{attribute 'linkalways'} 
{attribute 'no_explicit_call' := 'This FB is a CLASS and must be accessed using methods or properties'}
{attribute 'enable_dynamic_creation'}
FUNCTION_BLOCK Node_F_VN_MedianElementElementwise_SINT EXTENDS VisionNode
VAR
    ipContainer : _ITcVnContainer;
    nMedian : _SINT(0);
    hrPrev : _HRESULT(S_OK);
    hresult : _HRESULT(S_OK);
END_VAR

METHOD PUBLIC  Clone : I_Node
VAR
	pNode : POINTER TO Node_F_VN_MedianElementElementwise_SINT;
END_VAR
pNode := __NEW(Node_F_VN_MedianElementElementwise_SINT);
Clone := pNode^;
END_METHOD

METHOD FB_init : BOOL
VAR_INPUT
	bInitRetains : BOOL; // if TRUE, the retain variables are initialized (warm start / cold start)
	bInCopyCode : BOOL;  // if TRUE, the instance afterwards gets moved into the copy code (online change)
END_VAR
AddInput('ipContainer', ipContainer);
AddInput('nMedian', nMedian);
AddInput('hrPrev', hrPrev);
AddOutput('ipContainer', ipContainer);
AddOutput('hresult',hresult);
END_METHOD

METHOD PROTECTED OnExecute : HRESULT
hresult.Value := F_VN_MedianElementElementwise_SINT(
    ipContainer := ipContainer.Value,
    nMedian := nMedian.Value,
    hrPrev:= hrPrev.Value);
END_METHOD

METHOD PUBLIC PreExecutionCheck
VAR_INPUT
	Check : I_PreExecutionChecks;
END_VAR
Check.IsTrue(ipContainer.IsValid, 'ipContainer must be a valid container');
END_METHOD

END_FUNCTION_BLOCK

(* stored: Version 1.1.0.1, ProductVersion 3.1.4024.13
   POU Node_F_VN_MedianElementElementwise_SINT: Id {52d2e324-de06-49ab-9989-1c04961fd3e5}, SpecialFunc None
   Folder Constructor: Id {127eeb46-aa90-4fdd-a91a-40f4a0154d56}
   Method Clone: Id {ebb84139-2b9d-4d78-b9af-d477e3c759d1}
   Method FB_init: Id {c0e90acc-c089-402c-938f-d56400000201}
   Method OnExecute: Id {0e1c7eef-27de-4a68-8aa7-2292642b0ec9}
   Method PreExecutionCheck: Id {849d14e0-767a-43fa-8ac0-5db685ec12f6} *)
